INTERFACE I_SD_ValveState

METHOD Close : BOOL
VAR_INPUT
END_VAR
END_METHOD

METHOD Open : BOOL
VAR_INPUT
END_VAR
END_METHOD

METHOD RUN
END_METHOD

METHOD SetTransition
VAR_INPUT
    transition : I_Transitive;
END_VAR
END_METHOD

PROPERTY StateName : STRING
GET
END_GET
END_PROPERTY

END_INTERFACE

(* stored: Version 1.1.0.1, ProductVersion 3.1.4024.12
   Itf I_SD_ValveState: Id {11fc0dc5-5ce0-41f1-97b6-d259d310fbc8}
   Method Close: Id {e6e36200-c6b8-49d9-b173-3330708f4805}
   Method Open: Id {57dcb4a3-dc6a-45b8-b197-facbd22315ce}
   Method RUN: Id {5b82c0a1-23f7-4049-967b-5f7e149e495b}
   Method SetTransition: Id {dc246f6b-af9a-4b0b-8b87-5db27e4badfc}
   Property StateName: Id {a91f2d09-82e9-46d4-a25d-d3e08f17aa20}
   Get Get: Id {2799e6ce-9b32-41d0-a059-1cd8a3413a6b} *)
